FUNCTION AddMat3 : ARRAY[0..2, 0..2] OF LREAL
VAR_INPUT
	mat1: ARRAY[0..2, 0..2] OF REAL;
	mat2: ARRAY[0..2, 0..2] OF REAL;
END_VAR

VAR
	i, j: INT; 
END_VAR

FOR i := 0 TO 2 DO
	FOR j := 0 TO 2 DO
		AddMat3[i,j] := mat1[i,j] + mat2[i,j];
	END_FOR
END_FOR

END_FUNCTION

(* stored: Version 1.1.0.1, ProductVersion 3.1.4024.11
   POU AddMat3: Id {31e4cf46-7780-4daf-a11c-d89cf5ae93dd}, SpecialFunc None *)
